PROGRAM CFCPOU
VAR
	// Start Button
	btnStart: BOOL;
	// Stop Button
	btnStop: BOOL;
	// Motor Starter Coil
	Coil: BOOL;
END_VAR
VAR // added by the converter: edge detectors and wires of the graphical bodies
    _w1 : BOOL;
END_VAR

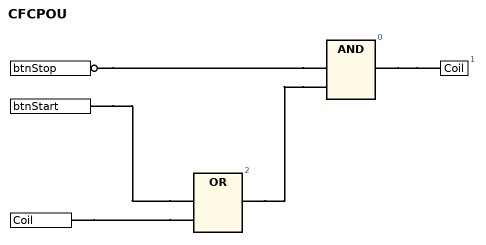
Coil := NOT btnStop AND _w1;
_w1 := btnStart OR Coil;

END_PROGRAM

(* stored: Version 1.1.0.1, ProductVersion 3.1.4024.15
   POU CFCPOU: Id {323a1b16-5dd3-4df2-aab8-81bf2bb9099f}, SpecialFunc None *)
